{attribute 'GeneratedUsingTerminal: EK1100-0000-0018'}
{attribute addProperty BoxType "EK1100-0000-0018"}
{attribute addProperty Id "Beckhoff_AMI8xxxEK1122Beckhoff_AMI8xxxEK1122_EC6540EE80"}
{attribute addProperty CRC "2092159243"}
{attribute addProperty Size "80"}
TYPE EK1100_Beckhoff_AMI8xxx_7CB3D10B EXTENDS EK1100_AB5A9467 :
STRUCT
	{attribute addProperty Name "Beckhoff_AMI8xxxEK1122"}
	Beckhoff_AMI8xxxEK1122 : Beckhoff_AMI8xxxEK1122_EC6540EE;
END_STRUCT
END_TYPE

(* stored: Version 1.2.0.0, ProductVersion 3.1.4024.9
   DUT EK1100_Beckhoff_AMI8xxx_7CB3D10B: Id {8e9702f7-99d1-4d8c-a403-4b1e36710193} *)
